// Mitsubishi GX Works2 project: BookEX3_7 DataType   PLC: Q13UDV

TYPE DateTime : STRUCT
  Year : INT;
  Month : INT;
  Day : INT;
  WeekDay : INT;
  iHour : INT;
  iMin : INT;
  iSec : INT;
  ms : INT;
END_STRUCT END_TYPE

TYPE Vector : STRUCT
  axisX : REAL;
  axisY : REAL;
  axisZ : REAL;
END_STRUCT END_TYPE

TYPE WordBit : STRUCT
  Data : DWORD;
  Flag : BOOL;
END_STRUCT END_TYPE

// global labels: Global
VAR_GLOBAL
  bVar0 AT M5000 : BOOL;
  abArray0 AT M5010 : ARRAY [0..49] OF BOOL;
  sStr0 AT D5000 : STRING[199];
  sStr1 AT D5100 : STRING[199];
  sStr2 AT D5200 : STRING[199];
  sStr3 AT D5300 : STRING[199];
  sStr4 AT D5400 : STRING[199];
  sStr5 AT D5500 : STRING[199];
  sStr6 AT D5600 : STRING[199];
  sStr7 AT D5700 : STRING[199];
  sStr8 AT D5800 : STRING[199];
  sStr9 AT D5900 : STRING[199];
  iVar0 AT D4500 : INT;
  iVar1 AT D4501 : INT;
  iVar2 AT D4502 : INT;
  iVar3 AT D4503 : INT;
  iVar4 AT D4504 : INT;
  iVar5 AT D4505 : INT;
  iVar6 AT D4506 : INT;
  iVar7 AT D4507 : INT;
  iVar8 AT D4508 : INT;
  iVar9 AT D4509 : INT;
  dVar0 AT D4510 : DINT;
  dVar1 AT D4512 : DINT;
  dVar2 AT D4514 : DINT;
  dVar3 AT D4516 : DINT;
  dVar4 AT D4518 : DINT;
  dVar5 AT D4520 : DINT;
  dVar6 AT D4522 : DINT;
  dVar7 AT D4524 : DINT;
  dVar8 AT D4526 : DINT;
  dVar9 AT D4528 : DINT;
  wVar0 AT D4530 : WORD;
  wVar1 AT D4531 : WORD;
  wVar2 AT D4532 : WORD;
  wVar3 AT D4533 : WORD;
  wVar4 AT D4534 : WORD;
  wVar5 AT D4535 : WORD;
  wVar6 AT D4536 : WORD;
  wVar7 AT D4537 : WORD;
  wVar8 AT D4538 : WORD;
  wVar9 AT D4539 : WORD;
  dwVar0 AT D4540 : DWORD;
  dwVar1 AT D4542 : DWORD;
  dwVar2 AT D4544 : DWORD;
  dwVar3 AT D4546 : DWORD;
  dwVar4 AT D4548 : DWORD;
  dwVar5 AT D4550 : DWORD;
  dwVar6 AT D4552 : DWORD;
  dwVar7 AT D4554 : DWORD;
  dwVar8 AT D4556 : DWORD;
  dwVar9 AT D4558 : DWORD;
  fsVar0 AT D4560 : REAL;
  fsVar1 AT D4562 : REAL;
  fsVar2 AT D4564 : REAL;
  fsVar3 AT D4566 : REAL;
  fsVar4 AT D4568 : REAL;
  fsVar5 AT D4570 : REAL;
  fsVar6 AT D4572 : REAL;
  fsVar7 AT D4574 : REAL;
  fsVar8 AT D4576 : REAL;
  fsVar9 AT D4578 : REAL;
  fdVar0 AT D4580 : LREAL;
  tTime0 AT D4620 : TIME;
  tTime1 AT D4622 : TIME;
  tTime2 AT D4624 : TIME;
  tTime3 AT D4626 : TIME;
  tTime4 AT D4628 : TIME;
  tTime5 AT D4630 : TIME;
  tTime6 AT D4632 : TIME;
  tTime7 AT D4634 : TIME;
  tTime8 AT D4636 : TIME;
  tTime9 AT D4638 : TIME;
  tTime10 AT D4640 : TIME;
  bVar1 AT M5001 : BOOL;
  bVar2 AT M5002 : BOOL;
  bVar3 AT M5003 : BOOL;
  bVar4 AT M5004 : BOOL;
  bVar5 AT M5005 : BOOL;
  bVar6 AT M5006 : BOOL;
  bVar7 AT M5007 : BOOL;
  bVar8 AT M5008 : BOOL;
  bVar9 AT M5009 : BOOL;
  abArray1 AT M5060 : ARRAY [0..49] OF BOOL;
  abArray2 AT M5110 : ARRAY [0..49] OF BOOL;
  abArray3 AT M5160 : ARRAY [0..49] OF BOOL;
  abArray4 AT M5210 : ARRAY [0..49] OF BOOL;
  abArray5 AT M5260 : ARRAY [0..49] OF BOOL;
  abArray6 AT M5310 : ARRAY [0..49] OF BOOL;
  abArray7 AT M5360 : ARRAY [0..49] OF BOOL;
  abArray8 AT M5410 : ARRAY [0..49] OF BOOL;
  abArray9 AT M5460 : ARRAY [0..49] OF BOOL;
  fdVar1 AT D4584 : LREAL;
  fdVar2 AT D4588 : LREAL;
  fdVar3 AT D4592 : LREAL;
  fdVar4 AT D4596 : LREAL;
  fdVar5 AT D4600 : LREAL;
  fdVar6 AT D4604 : LREAL;
  fdVar7 AT D4608 : LREAL;
  fdVar8 AT D4612 : LREAL;
  fdVar9 AT D4616 : LREAL;
  aSendData1 AT D100 : ARRAY [0..9] OF INT;
  aiTxData AT D4000 : ARRAY [0..99] OF INT;
  aiRxData AT D4100 : ARRAY [0..99] OF INT;
  iOpenOK AT D3900 : INT;
  iOpenERR AT D3901 : INT;
  iSendOK AT D3902 : INT;
  iSendERR AT D3903 : INT;
  iCloseOK AT D3906 : INT;
  iCloseERR AT D3907 : INT;
  iRecvOK AT D3904 : INT;
  iRecvERR AT D3905 : INT;
  aiTxData2 AT D4200 : ARRAY [0..99] OF INT;
  aiRxData2 AT D4300 : ARRAY [0..99] OF INT;
  iOpenOK2 AT D3908 : INT;
  iOpenERR2 AT D3909 : INT;
  iSendOK2 AT D3910 : INT;
  iSendERR2 AT D3911 : INT;
  iRecvOK2 AT D3912 : INT;
  iRecvERR2 AT D3913 : INT;
  iCloseOK2 AT D3914 : INT;
  iCloseERR2 AT D3915 : INT;
  iEOpenComp AT D3916 : INT;
  iEOpenReq AT D3917 : INT;
  iERecvFlag AT D3918 : INT;
  iOpenCode AT D3919 : INT;
  iSendCode AT D3920 : INT;
  iRecvCode AT D3921 : INT;
  iCloseCode AT D3922 : INT;
  iOpenCode2 AT D3923 : INT;
  iSendCode2 AT D3924 : INT;
  iRecvCode2 AT D3925 : INT;
  iCloseCode2 AT D3926 : INT;
  aRecvData1 AT D110 : ARRAY [0..9] OF INT;
  aSendData2 AT D120 : ARRAY [0..9] OF INT;
  aRecvData2 AT D130 : ARRAY [0..9] OF INT;
END_VAR
// user libraries (not included): HMI

PROGRAM ExArray
VAR
  aBoxNo1 : ARRAY [0..99] OF INT;
  aBoxNo2 : ARRAY [0..99,0..99] OF INT;
  aBoxNo3 : ARRAY [0..9,0..9,0..9] OF INT;
  aStr1 : ARRAY [1..9] OF STRING[199] := [9('')];
  aStr2 : ARRAY [1..9,1..9] OF STRING[32] := [81('')];
  aStr3 : ARRAY [1..9,1..9,0..9] OF STRING[32] := [810('')];
  aStatus1 : ARRAY [0..4] OF WORD;
  aStatus2 : ARRAY [0..4,1..5] OF WORD;
  aStatus3 : ARRAY [0..4,1..5,2..6] OF WORD;
  aVector1 : ARRAY [0..4] OF Vector;
  aVector2 : ARRAY [0..4,0..3] OF Vector;
  aVector3 : ARRAY [0..4,0..3,0..2] OF Vector;
  bLabel1 : ARRAY [0..3] OF BOOL;
  bLabel2 : ARRAY [0..4,0..3] OF BOOL;
  bLabel3 : ARRAY [0..5,0..4,0..3] OF BOOL;
  aiNo : ARRAY [0..99] OF INT;
  aiSno : ARRAY [0..99] OF INT;
END_VAR
(* structured ladder/FBD written out as ST: instructions are called as NAME(EN, inputs, outputs); _pN, _eN, _tN stand for wires *)
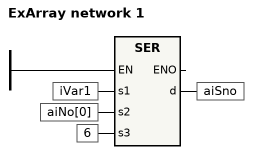
(* network 1 *)
SER(TRUE, iVar1, aiNo[0], 6, aiSno);
END_PROGRAM

PROGRAM ExDataType
VAR
  Mov4WORD_1 : Mov4WORD;
  Mov8WORD_1 : Mov8WORD;
END_VAR
(* structured ladder/FBD written out as ST: instructions are called as NAME(EN, inputs, outputs); _pN, _eN, _tN stand for wires *)
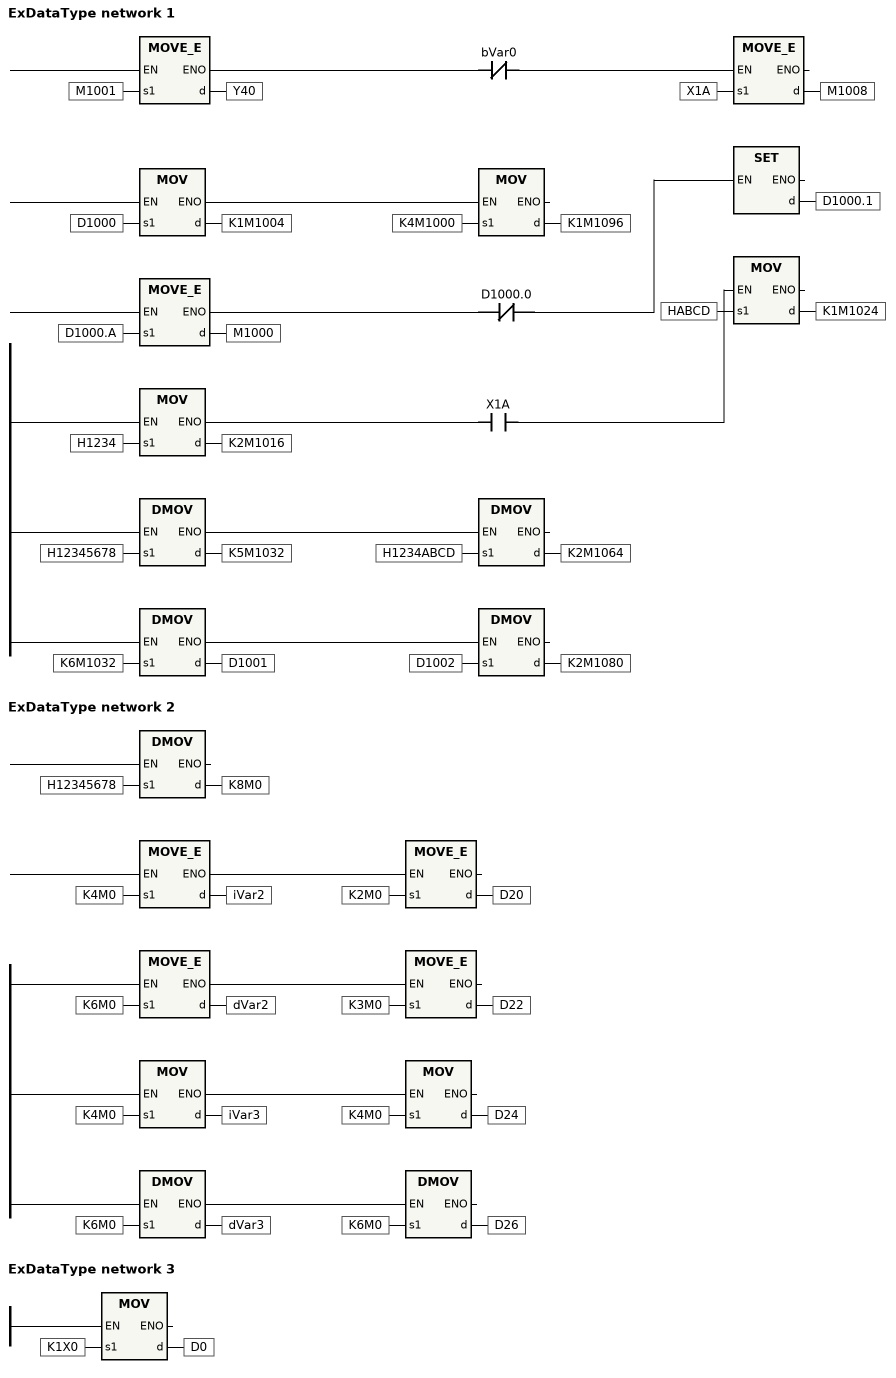
(* network 1 *)
_e1 := MOVE_E(TRUE, M1001, Y40);
MOVE_E(_e1 AND NOT bVar0, X1A, M1008);
_e2 := MOVE_E(TRUE, D1000.A, M1000);
SET(_e2 AND NOT D1000.0, D1000.1);
_e3 := MOV(TRUE, H1234, K2M1016);
MOV(_e3 AND X1A, HABCD, K1M1024);
_e4 := MOV(TRUE, D1000, K1M1004);
MOV(_e4, K4M1000, K1M1096);
_e5 := DMOV(TRUE, H12345678, K5M1032);
DMOV(_e5, H1234ABCD, K2M1064);
_e6 := DMOV(TRUE, K6M1032, D1001);
DMOV(_e6, D1002, K2M1080);
(* network 2 *)
DMOV(TRUE, H12345678, K8M0);
_e1 := MOVE_E(TRUE, K4M0, iVar2);
MOVE_E(_e1, K2M0, D20);
_e2 := MOVE_E(TRUE, K6M0, dVar2);
MOVE_E(_e2, K3M0, D22);
_e3 := MOV(TRUE, K4M0, iVar3);
MOV(_e3, K4M0, D24);
_e4 := DMOV(TRUE, K6M0, dVar3);
DMOV(_e4, K6M0, D26);
(* network 3 *)
MOV(TRUE, K1X0, D0);
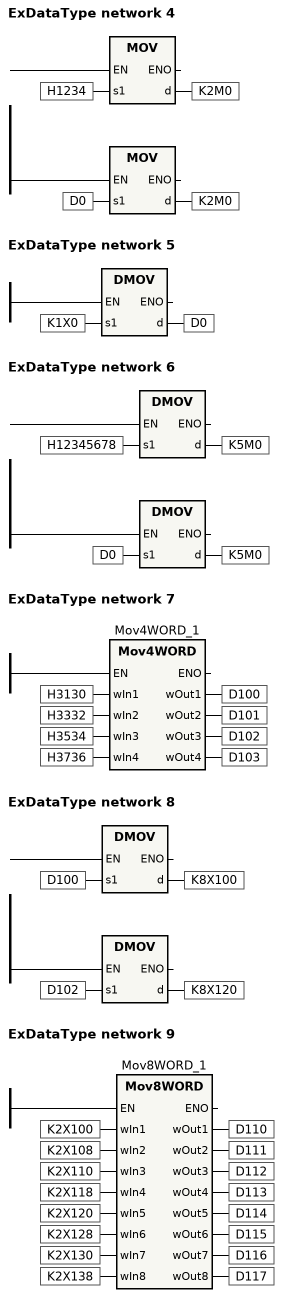
(* network 4 *)
MOV(TRUE, H1234, K2M0);
MOV(TRUE, D0, K2M0);
(* network 5 *)
DMOV(TRUE, K1X0, D0);
(* network 6 *)
DMOV(TRUE, H12345678, K5M0);
DMOV(TRUE, D0, K5M0);
(* network 7 *)
Mov4WORD_1(EN := TRUE, wIn1 := H3130, wIn2 := H3332, wIn3 := H3534, wIn4 := H3736, wOut1 => D100, wOut2 => D101, wOut3 => D102, wOut4 => D103);
(* network 8 *)
DMOV(TRUE, D100, K8X100);
DMOV(TRUE, D102, K8X120);
(* network 9 *)
Mov8WORD_1(EN := TRUE, wIn1 := K2X100, wIn2 := K2X108, wIn3 := K2X110, wIn4 := K2X118, wIn5 := K2X120, wIn6 := K2X128, wIn7 := K2X130, wIn8 := K2X138, wOut1 => D110, wOut2 => D111, wOut3 => D112, wOut4 => D113, wOut5 => D114, wOut6 => D115, wOut7 => D116, wOut8 => D117);
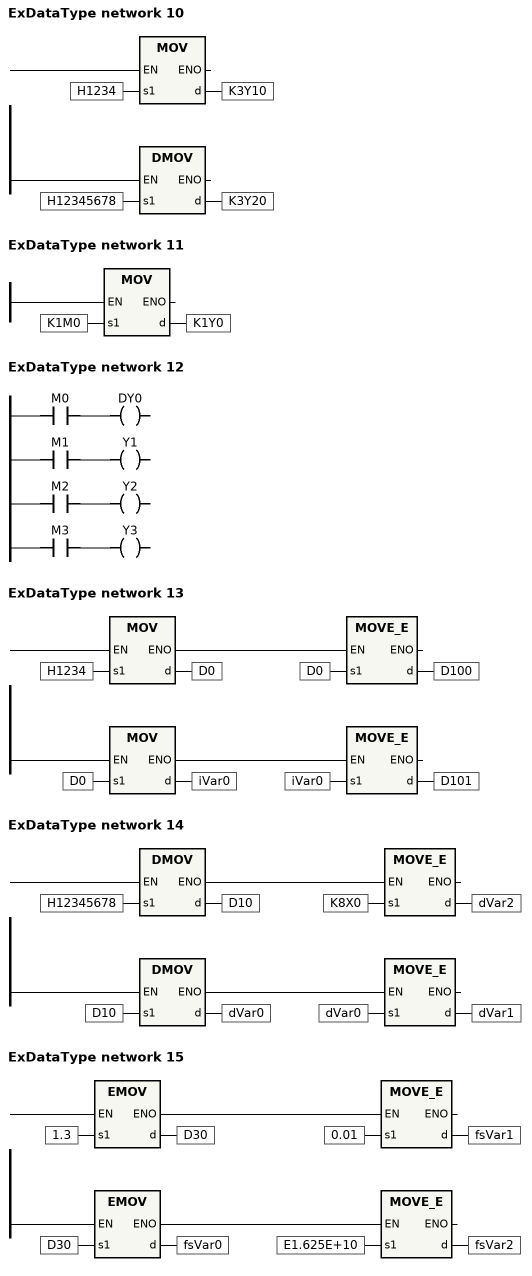
(* network 10 *)
MOV(TRUE, H1234, K3Y10);
DMOV(TRUE, H12345678, K3Y20);
(* network 11 *)
MOV(TRUE, K1M0, K1Y0);
(* network 12 *)
DY0 := M0;
Y1 := M1;
Y2 := M2;
Y3 := M3;
(* network 13 *)
_e1 := MOV(TRUE, H1234, D0);
MOVE_E(_e1, D0, D100);
_e2 := MOV(TRUE, D0, iVar0);
MOVE_E(_e2, iVar0, D101);
(* network 14 *)
_e1 := DMOV(TRUE, H12345678, D10);
MOVE_E(_e1, K8X0, dVar2);
_e2 := DMOV(TRUE, D10, dVar0);
MOVE_E(_e2, dVar0, dVar1);
(* network 15 *)
_e1 := EMOV(TRUE, 1.3, D30);
MOVE_E(_e1, 0.01, fsVar1);
_e2 := EMOV(TRUE, D30, fsVar0);
MOVE_E(_e2, E1.625E+10, fsVar2);
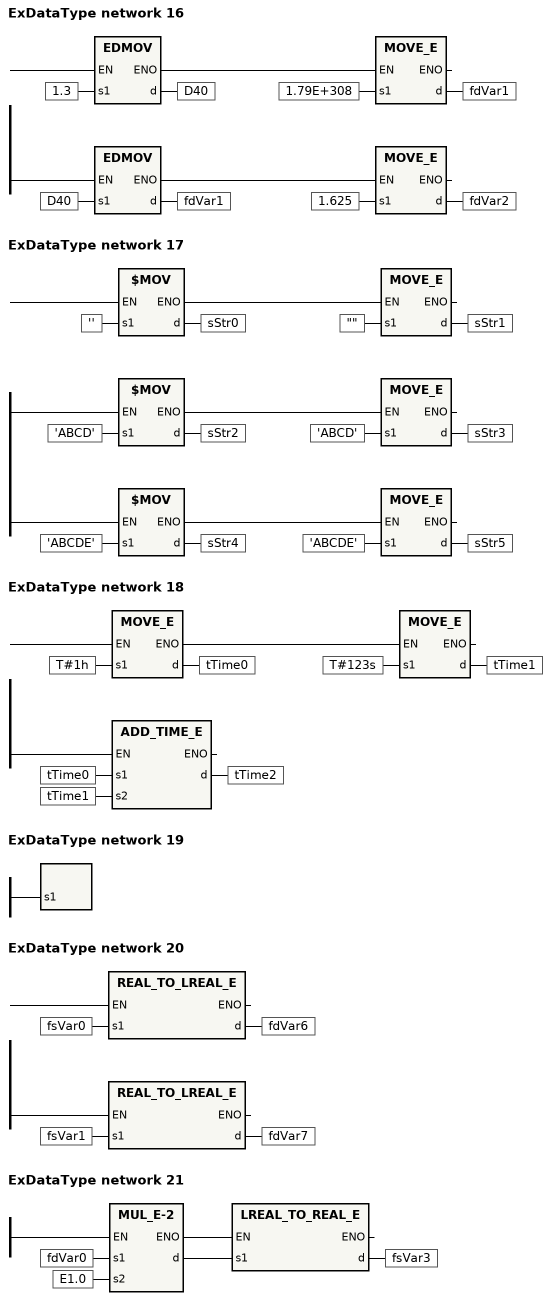
(* network 16 *)
_e1 := EDMOV(TRUE, 1.3, D40);
MOVE_E(_e1, 1.79E+308, fdVar1);
_e2 := EDMOV(TRUE, D40, fdVar1);
MOVE_E(_e2, 1.625, fdVar2);
(* network 17 *)
_e1 := $MOV(TRUE, '', sStr0);
MOVE_E(_e1, "", sStr1);
_e2 := $MOV(TRUE, 'ABCD', sStr2);
MOVE_E(_e2, 'ABCD', sStr3);
_e3 := $MOV(TRUE, 'ABCDE', sStr4);
MOVE_E(_e3, 'ABCDE', sStr5);
(* network 18 *)
_e1 := MOVE_E(TRUE, T#1h, tTime0);
MOVE_E(_e1, T#123s, tTime1);
ADD_TIME_E(TRUE, tTime0, tTime1, tTime2);
(* network 19 *)
(* element kind 10  <- TRUE *)
(* network 20 *)
REAL_TO_LREAL_E(TRUE, fsVar0, fdVar6);
REAL_TO_LREAL_E(TRUE, fsVar1, fdVar7);
(* network 21 *)
_e2 := MUL_E(TRUE, fdVar0, E1.0, _t1);
LREAL_TO_REAL_E(_e2, _t1, fsVar3);
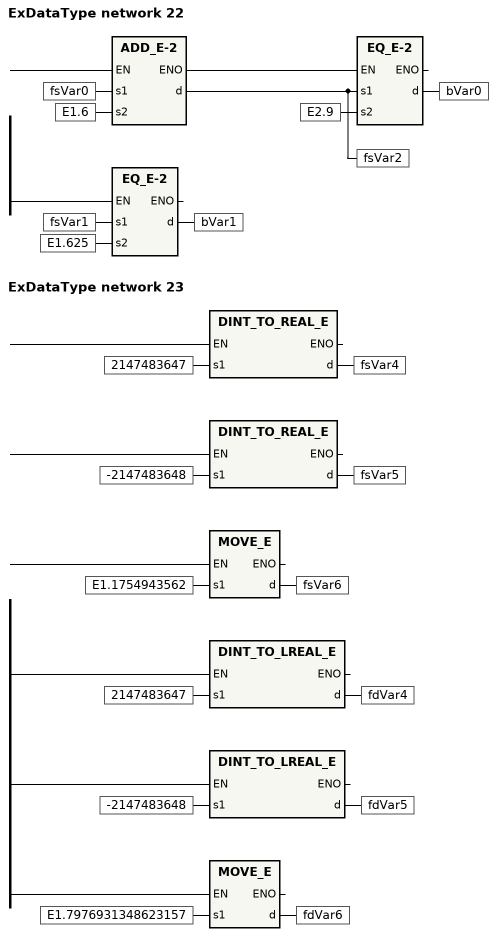
(* network 22 *)
_e1 := ADD_E(TRUE, fsVar0, E1.6, fsVar2);
EQ_E(_e1, fsVar2, E2.9, bVar0);
EQ_E(TRUE, fsVar1, E1.625, bVar1);
(* network 23 *)
DINT_TO_REAL_E(TRUE, 2147483647, fsVar4);
DINT_TO_REAL_E(TRUE, -2147483648, fsVar5);
MOVE_E(TRUE, E1.1754943562, fsVar6);
DINT_TO_LREAL_E(TRUE, 2147483647, fdVar4);
DINT_TO_LREAL_E(TRUE, -2147483648, fdVar5);
MOVE_E(TRUE, E1.7976931348623157, fdVar6);
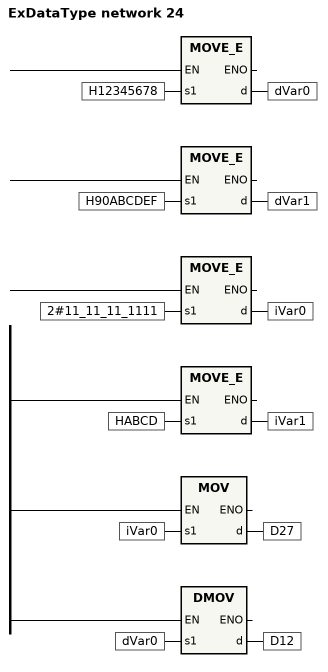
(* network 24 *)
MOVE_E(TRUE, H12345678, dVar0);
MOVE_E(TRUE, H90ABCDEF, dVar1);
MOVE_E(TRUE, 2#11_11_11_1111, iVar0);
MOVE_E(TRUE, HABCD, iVar1);
MOV(TRUE, iVar0, D27);
DMOV(TRUE, dVar0, D12);
END_PROGRAM

PROGRAM ExReal
(* structured ladder/FBD written out as ST: instructions are called as NAME(EN, inputs, outputs); _pN, _eN, _tN stand for wires *)
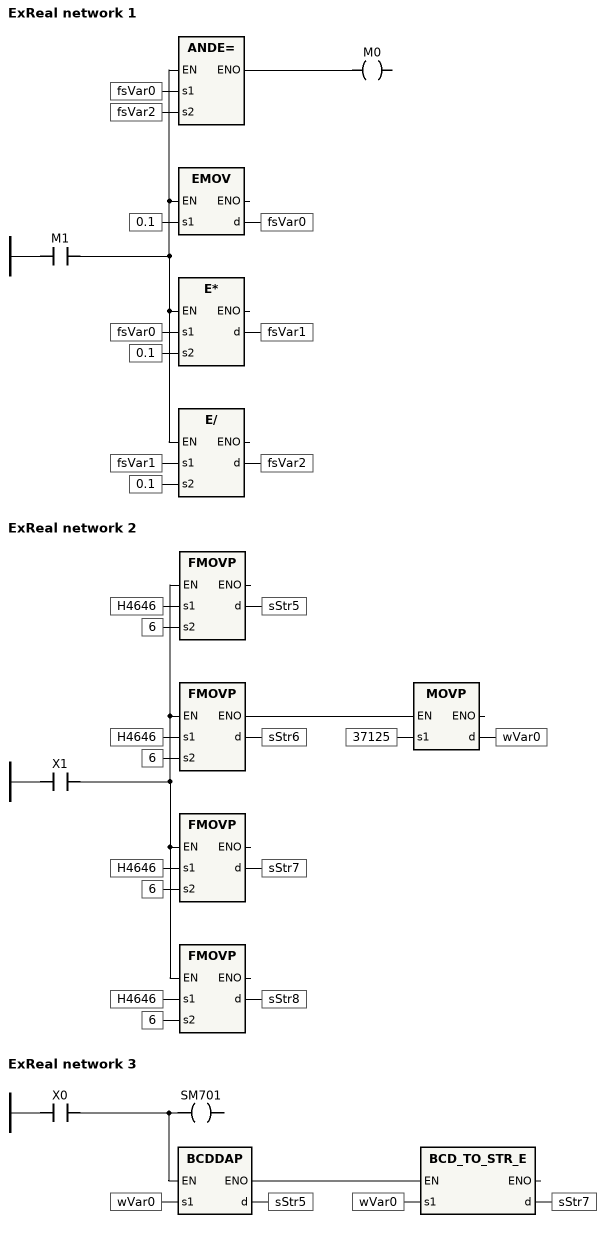
(* network 1 *)
EMOV(M1, 0.1, fsVar0);
E*(M1, fsVar0, 0.1, fsVar1);
E/(M1, fsVar1, 0.1, fsVar2);
_e1 := ANDE=(M1, fsVar0, fsVar2);
M0 := _e1;
(* network 2 *)
FMOVP(X1, H4646, 6, sStr5);
_e1 := FMOVP(X1, H4646, 6, sStr6);
MOVP(_e1, 37125, wVar0);
FMOVP(X1, H4646, 6, sStr7);
FMOVP(X1, H4646, 6, sStr8);
(* network 3 *)
SM701 := X0;
_e1 := BCDDAP(X0, wVar0, sStr5);
BCD_TO_STR_E(_e1, wVar0, sStr7);
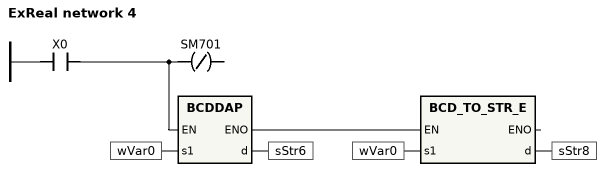
(* network 4 *)
SM701 := NOT X0;
_e1 := BCDDAP(X0, wVar0, sStr6);
BCD_TO_STR_E(_e1, wVar0, sStr8);
END_PROGRAM
